(* CoDeSys 2.3 export: ST_PSX_VALVE_OUT.EXP *)

(* Data type *)
TYPE ST_PSX_VALVE_OUT :
STRUCT
	Control  : UINT;
	SetPoint : INT;

END_STRUCT
END_TYPE
